// TwinCAT 3 PLC project MAS418_PLC
// ProgramVersion: 3.1.4023.0
// libraries:
//   Tc2_Standard, * (Beckhoff Automation GmbH)
//   Tc2_System, * (Beckhoff Automation GmbH)
//   Tc3_Module, * (Beckhoff Automation GmbH)
//   VisuDialogs, * (System)
// project tree:
//   / GlobalTextList.TcGTLO, PlcTask.TcTTO, Visualization Manager.TcVMO (not stored)
//   POUs/ MAIN.TcPOU
//   VISUs/ HMI.TcVIS
// real-time tasks:
//   TASK PlcTask: cycle T#10ms, priority 20, ADS port 350

CONFIGURATION MAS418_PLC
    RESOURCE PLC ON TwinCAT3
        TASK PlcTask(INTERVAL := T#10ms, PRIORITY := 20);
        PROGRAM MAIN WITH PlcTask : MAIN;
    END_RESOURCE
END_CONFIGURATION

// ---- POUs/MAIN.TcPOU
PROGRAM MAIN
VAR
		bStart  :BOOL;
		bEnable :BOOL;
		nINT : INT := -32768;
	    nUINT : UINT := 65535;
	    fREAL : REAL := 255.255;
		sPowerStatus: STRING := 'Power Off'; 
		nFloatConversion:INT;
		fFloatConversion:LREAL;
END_VAR

bEnable:= bStart;
fFloatConversion:=INT_TO_LREAL(nFloatConversion);

END_PROGRAM

// ---- GlobalTextList.TcGTLO
TEXTLIST GlobalTextList
  800 = '                  '
  66 = '%f'
  133 = '%i'
  154 = '%s'
  718 = 'Bool'
  689 = 'DataType Testing'
  0 = 'i'
  495 = 'INT'
  731 = 'Label'
  232 = 'Power On'
  628 = 'Power ON'
  206 = 'REAL'
  601 = 'STRING'
  522 = 'UINT'
END_TEXTLIST

// ---- VISUs/HMI.TcVIS
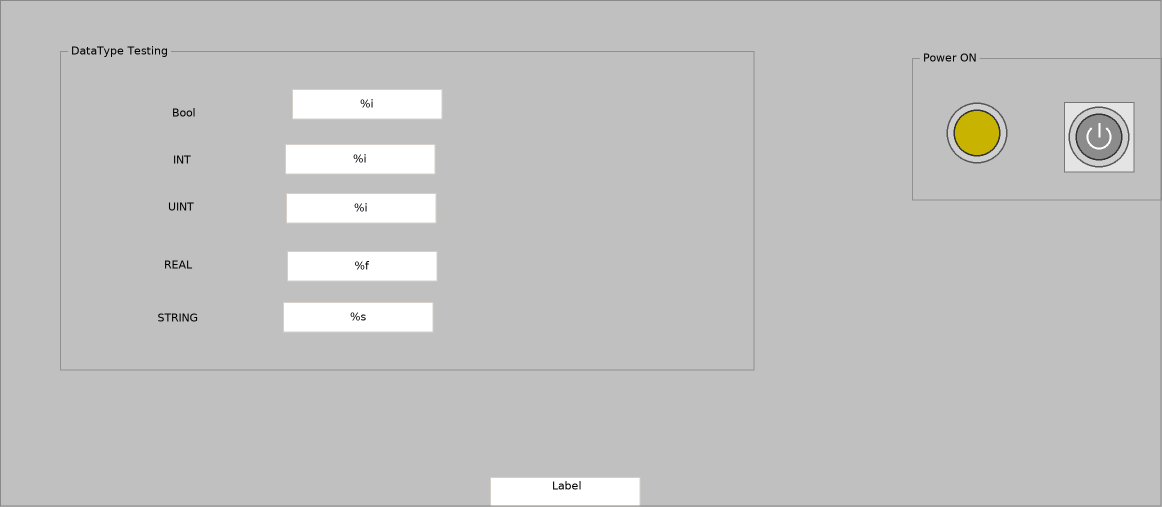
VISUALIZATION HMI  // 1162x507
    GroupBox (912,50 250x150), "Power ON"
        Lamp1 (30,48 70x70), variable: MAIN.bEnable, style: Lamp-Lamp1-Yellow
        PowerSwitch (152,52 70x70), variable: MAIN.bStart, behaviour: TOGGLE, style: Switch-PowerSwitch-Gray
    GroupBox (60,43 694x327), "DataType Testing"
        Textfield (223,259 150x30), "%s", text variable: MAIN.sPowerStatus
            OnMouseDown: write the text variable via Default
        Textfield (232,46 150x30), "%i", text variable: MAIN.bEnable
        Textfield (225,101 150x30), "%i", text variable: MAIN.nINT
        Textfield (226,150 150x30), "%i", text variable: MAIN.nUINT
        Textfield (227,208 150x30), "%f", text variable: MAIN.fREAL
        Label (49,55 150x30), "Bool"
        Label (47,102 150x30), "INT"
        Label (46,149 150x30), "UINT"
        Label (43,207 150x30), "REAL"
        Label (43,260 150x30), "STRING"
    Textfield (490,477 150x30)
    Label (492,471 150x30), "Label"
END_VISUALIZATION
